PROGRAM IOParams
VAR
	iForLoopDMXI1			: INT;
	iForLoopDMXI2			: INT;
	iForLoopDMXI3			: INT;
	iForLoopDMXI4			: INT;
	iForLoopDMXI5			: INT;
	iForLoopDMXI6			: INT;
	iForLoopDMXI7			: INT;
	iForLoopDMXI8			: INT;
	uiForLoopDMXI10			: UINT;
	uiForLoopDMXI11			: UINT;
	uiForLoopDebouncePNP	: UINT;
	uiForLoopDebounceNPN	: UINT;
END_VAR

//Link all the user-specified params to the respective Function Blocks
//RED

(*
RGB PARAMETERS - Hence, the Groups of 4 incremented in this way;

FOR iForLoopDMXI1:= 0 TO gc.uiMaxNrOfDMXChannel BY 4 DO
	g_ast.DMX[iForLoopDMXI1].I.ENWaveform		:= ENUM_I_Waveform.EN_Sin; //"50% duty cycle"
	g_ast.DMX[iForLoopDMXI1].I.fDutyCycle		:= 50; // %
	g_ast.DMX[iForLoopDMXI1].I.fLevel			:= iSlider5; //%
	g_ast.DMX[iForLoopDMXI1].I.fOffset			:= 0; // %
	g_ast.DMX[iForLoopDMXI1].I.usiBitDepth		:= 8; // 0-8, or 0-16, depending
	g_ast.DMX[iForLoopDMXI1].I.fPhase			:= 0; // %
	g_ast.DMX[iForLoopDMXI1].I.fDelay			:= 0; // %
	g_ast.DMX[iForLoopDMXI1].I.usiDelayDiv		:= 0; // which step to have delay applied
END_FOR

//GREEN
FOR iForLoopDMXI2:= 1 TO gc.uiMaxNrOfDMXChannel BY 4 DO
	g_ast.DMX[iForLoopDMXI2].I.ENWaveform		:= ENUM_I_Waveform.EN_Sin; //"50% duty cycle"
	g_ast.DMX[iForLoopDMXI2].I.fDutyCycle		:= 50; // %
	g_ast.DMX[iForLoopDMXI2].I.fLevel			:= iSlider6; //%
	g_ast.DMX[iForLoopDMXI2].I.fOffset			:= 0; // %
	g_ast.DMX[iForLoopDMXI2].I.usiBitDepth		:= 8; // 0-8, or 0-16, depending
	g_ast.DMX[iForLoopDMXI2].I.fPhase			:= 0; // %
	g_ast.DMX[iForLoopDMXI2].I.fDelay			:= 0; // %
	g_ast.DMX[iForLoopDMXI2].I.usiDelayDiv		:= 0; // which step to have delay applied
END_FOR

//BLUE
FOR iForLoopDMXI3:= 2 TO gc.uiMaxNrOfDMXChannel BY 4 DO
	g_ast.DMX[iForLoopDMXI3].I.ENWaveform		:= ENUM_I_Waveform.EN_Sin; //"50% duty cycle"
	g_ast.DMX[iForLoopDMXI3].I.fDutyCycle		:= 50; // %
	g_ast.DMX[iForLoopDMXI3].I.fLevel			:= iSlider7; //%
	g_ast.DMX[iForLoopDMXI3].I.fOffset			:= 0; // %
	g_ast.DMX[iForLoopDMXI3].I.usiBitDepth		:= 8; // 0-8, or 0-16, depending
	g_ast.DMX[iForLoopDMXI3].I.fPhase			:= 0; // %
	g_ast.DMX[iForLoopDMXI3].I.fDelay			:= 0; // %
	g_ast.DMX[iForLoopDMXI3].I.usiDelayDiv		:= 0; // which step to have delay applied
END_FOR

//WHITE
FOR iForLoopDMXI4:= 3 TO gc.uiMaxNrOfDMXChannel BY 4 DO
	g_ast.DMX[iForLoopDMXI4].I.ENWaveform		:= ENUM_I_Waveform.EN_Sin; //"50% duty cycle"
	g_ast.DMX[iForLoopDMXI4].I.fDutyCycle		:= 50; // %
	g_ast.DMX[iForLoopDMXI4].I.fLevel			:= iSlider8; //%
	g_ast.DMX[iForLoopDMXI4].I.fOffset			:= 0; // %
	g_ast.DMX[iForLoopDMXI4].I.usiBitDepth		:= 8; // 0-8, or 0-16, depending
	g_ast.DMX[iForLoopDMXI4].I.fPhase			:= 0; // %
	g_ast.DMX[iForLoopDMXI4].I.fDelay			:= 0; // %
	g_ast.DMX[iForLoopDMXI4].I.usiDelayDiv		:= 0; // which step to have delay applied
END_FOR


FOR iForLoopDMXI5	:= 0 TO gc.uiMaxNrOfDMXChannel BY 4 DO 
	g_ast.DMX[iForLoopDMXI5].I.fFrequency		:= iSlider1; //Hz
END_FOR

FOR iForLoopDMXI6	:= 0 TO gc.uiMaxNrOfDMXChannel BY 4 DO 
	g_ast.DMX[iForLoopDMXI6].I.fFrequency		:= iSlider2; //Hz
END_FOR

FOR iForLoopDMXI7	:= 0 TO gc.uiMaxNrOfDMXChannel BY 4 DO 
	g_ast.DMX[iForLoopDMXI7].I.fFrequency		:= iSlider3; //Hz
END_FOR

FOR iForLoopDMXI8	:= 0 TO gc.uiMaxNrOfDMXChannel BY 4 DO 
	g_ast.DMX[iForLoopDMXI8].I.fFrequency		:= iSlider4; //Hz
END_FOR
*)

FOR uiForLoopDMXI10:= 0 TO gc.uiDUTConfigCountSplit BY 1 DO
	g_ast.DMX[uiForLoopDMXI10].I.fFrequency		:= 0;
	g_ast.DMX[uiForLoopDMXI10].I.ENWaveform		:= ENUM_I_Waveform.EN_GateCtrl;
	g_ast.DMX[uiForLoopDMXI10].I.ENValRange		:= ENUM_I_ValRange.EN_8Bit;
	g_ast.DMX[uiForLoopDMXI10].I.fDutyCycle		:= 100; // %
	g_ast.DMX[uiForLoopDMXI10].I.fLevel			:= 100; //%
	g_ast.DMX[uiForLoopDMXI10].I.fOffset		:= 0; // %
	g_ast.DMX[uiForLoopDMXI10].I.usiBitDepth	:= 8; // 0-8, or 0-16, depending
	g_ast.DMX[uiForLoopDMXI10].I.fPhase			:= 0; // %
	g_ast.DMX[uiForLoopDMXI10].I.fDelay			:= 0; // %
	g_ast.DMX[uiForLoopDMXI10].I.usiDelayDiv	:= 0; // which step to have delay applied
//Channels for Configuration of testing on other DMX Channels;
END_FOR

FOR uiForLoopDMXI10:= gc.uiChannelSplitCount TO gc.uiMaxNrOfDMXChannel BY 1 DO
	g_ast.DMX[uiForLoopDMXI10].I.fFrequency		:= 0;
	g_ast.DMX[uiForLoopDMXI10].I.ENWaveform		:= ENUM_I_Waveform.EN_GateConfig;
	g_ast.DMX[uiForLoopDMXI10].I.ENValRange		:= ENUM_I_ValRange.EN_8Bit;
	g_ast.DMX[uiForLoopDMXI10].I.fDutyCycle		:= 100; // %
	g_ast.DMX[uiForLoopDMXI10].I.fLevel			:= 100; //%
	g_ast.DMX[uiForLoopDMXI10].I.fOffset		:= 0; // %
	g_ast.DMX[uiForLoopDMXI10].I.usiBitDepth	:= 8; // 0-8, or 0-16, depending
	g_ast.DMX[uiForLoopDMXI10].I.fPhase			:= 0; // %
	g_ast.DMX[uiForLoopDMXI10].I.fDelay			:= 0; // %
	g_ast.DMX[uiForLoopDMXI10].I.usiDelayDiv	:= 0; // which step to have delay applied
//Channels for Configuration of testing on other DMX Channels;
END_FOR

//Input Debounce Params PNP
FOR uiForLoopDebouncePNP	:= 0 TO gc.uiMaxNrDMXTestCh BY 1 DO
	g_ast.arrFBIntPNP[uiForLoopDebouncePNP].I.tOnDelay	:= T#0S;
	g_ast.arrFBIntPNP[uiForLoopDebouncePNP].I.tOffDelay	:= T#10MS;
END_FOR

//Input Debounce Params NPN
FOR uiForLoopDebounceNPN	:= 0 TO gc.uiMaxNrDMXTestCh BY 1 DO
	g_ast.arrFBIntNPN[uiForLoopDebounceNPN].I.tOnDelay	:= T#0S;
	g_ast.arrFBIntNPN[uiForLoopDebounceNPN].I.tOffDelay	:= T#3MS;
END_FOR

//Read the CSV Parameters into the DMX FBs - via the "mediating" Config arrays
FOR uiForLoopDMXI11:= 0 TO gc.uiMaxNrOfDMXChannel BY 1 DO
	g_ast.DMX[DMXTest.arr_uiRecipeIndex[uiForLoopDMXI11]].I.usiInputConfig	:= 	DMXTest.arr_usiRecipeSetting[uiForLoopDMXI11];
END_FOR

END_PROGRAM

(* stored: Version 1.1.0.1, ProductVersion 3.1.4024.6
   POU IOParams: Id {a5664a88-4512-4669-bbf3-ce5ec238c33e}, SpecialFunc None *)
